// TIA Portal V17 export
// export: Created 2024-08-07T21:44:03.4611767Z, ExportSetting WithDefaults, DisplayName Totally Integrated Automation Portal, DisplayVersion V17 Update 7, DisplayName TIA Portal Openness, DisplayVersion V17 Update 7, DisplayName TIA Portal Version Control Interface, DisplayVersion V17, DisplayName SINAMICS Startdrive Advanced, DisplayVersion V17 SP2, DisplayName SINAMICS Startdrive G110M, G120, G120C, G120D, G120P, G115D, DisplayVersion V17 SP2, DisplayName SINAMICS Startdrive G130, G150, S120, S150, SINAMICS MV, S210, DisplayVersion V17 SP2, DisplayName STEP 7 Professional, DisplayVersion V17 Update 7, DisplayName STEP 7 Safety, DisplayVersion V17 Update 6, DisplayName WinCC Advanced / Unified PC, DisplayVersion V17 Update 7
DATA_BLOCK "DB_ProductionCountersEdit"   // DB66
{ S7_Optimized_Access := 'TRUE' }
VERSION : 0.1
// stored: AutoNumber true, DBAccessibleFromOPCUA true, DBAccessibleFromWebserver true, IsOnlyStoredInLoadMemory false, IsRetainMemResEnabled false, IsWriteProtectedInAS false, MemoryReserve 100
   VAR
      ProgramNumber : Int := 1;
      ProgramName : String[50] := '2569703X-LH';
      ProductCounters { S7_SetPoint := 'True'} : "UDT_ProductionProgramCounters";
      SettingsCanBeChanged : Bool := FALSE;
      DeleteCounters : Int := 0;
   END_VAR
BEGIN
   ProductCounters.Product[1].Shift[1..3].Ok := 0;
   ProductCounters.Product[2].Shift[1..3].Ok := 0;
   ProductCounters.Product[3].Shift[1..3].Ok := 0;
   ProductCounters.Product[4].Shift[1..3].Ok := 0;
   ProductCounters.Product[5].Shift[1..3].Ok := 0;
   ProductCounters.Product[6].Shift[1..3].Ok := 0;
   ProductCounters.Product[7].Shift[1..3].Ok := 0;
   ProductCounters.Product[8].Shift[1..3].Ok := 0;
   ProductCounters.Product[1].Shift[1..3].Nok := 0;
   ProductCounters.Product[2].Shift[1..3].Nok := 0;
   ProductCounters.Product[3].Shift[1..3].Nok := 0;
   ProductCounters.Product[4].Shift[1..3].Nok := 0;
   ProductCounters.Product[5].Shift[1..3].Nok := 0;
   ProductCounters.Product[6].Shift[1..3].Nok := 0;
   ProductCounters.Product[7].Shift[1..3].Nok := 0;
   ProductCounters.Product[8].Shift[1..3].Nok := 0;
   ProductCounters.Product[1..8].Overall.Ok := 0;
   ProductCounters.Product[1..8].Overall.Nok := 0;
END_DATA_BLOCK
